// TwinCAT 3 PLC project PLC
// ProgramVersion: 3.1.4024.0
// libraries:
//   SPT Base Types, * (Beckhoff Automation LLC)
//   SPT Components, * (Beckhoff Automation LLC)
//   SPT Motion Control, * (Beckhoff Automation LLC)
//   Tc2_MC2, * (Beckhoff Automation GmbH)
//   Tc2_MC2_Drive, * (Beckhoff Automation GmbH)
//   Tc2_Standard, * (Beckhoff Automation GmbH)
//   Tc2_System, * (Beckhoff Automation GmbH)
//   Tc3_Module, * (Beckhoff Automation GmbH)
//   Tc3_PackML_V2, * (Beckhoff Automation GmbH)
//   VisuDialogs, * (System)
// project tree:
//   / GlobalTextList.TcGTLO, PlcTask.TcTTO, Visualization Manager.TcVMO (not stored)
//   POUs/ MAIN.TcPOU
//   VISUs/ VIS_Main.TcVIS (not stored)
//   _Machine/00_Machine/ FB_UM_Machine.TcPOU
//   _Machine/VISUs/VFMs/ VFM_Machine.TcVIS (not stored), VFM_MachineControl.TcVIS (not stored), VFM_Module.TcVIS (not stored), VFM_OperatingMode.TcVIS (not stored), VFM_PackML.TcVIS (not stored), VFM_PackML_Manual.TcVIS (not stored)
//   _Machine/_Components/Drives/AX5000/ FB_Drive_AX5000.TcPOU, I_Drive_AX5000.TcIO
//   _Machine/_Components/Misc/ FB_StatFilter.TcPOU (not stored), F_TaskTime.TcPOU (not stored)
//   _Machine/_Components/TempController/DUTs/ ST_HMI_TempController.TcDUT (not stored), ST_HMI_TempController_Command.TcDUT (not stored), ST_HMI_TempController_Config.TcDUT (not stored), ST_HMI_TempController_Status.TcDUT (not stored), ST_Param_TempController.TcDUT (not stored)
//   _Machine/_Components/TempController/ FB_TempController.TcPOU, FB_TempCtrl.TcPOU (not stored), I_TemperatureController.TcIO (not stored)
//   _Machine/_Components/TempController/VISUs/VFMs/ VFM_TempController.TcVIS (not stored)
//   _Machine/_Components/TempController/VISUs/ VIS_TempCtrl.TcVIS (not stored)
// real-time tasks:
//   TASK PlcTask: cycle T#10ms, priority 20, ADS port 350
// motion (NC):
//   TASK NC-Task 1 SAF: cycle T#2ms, priority 4, ADS port 501
//   TASK NC-Task 1 SVB: cycle T#10ms, priority 8, ADS port 511
//   AXIS Axis 1 (id 1)
//     OtherSettings: AllowMotionCmdToSlave=true
//     encoder EncType=8
//       EncPara: MaxCount=#x0036ee7f
//     drive DrvType=9
//       DrvPara: MaxCount=#xffffffff, DriveControlDWord=#x00000100
//         Analog: VeloScale=6, TorqueSetpointScale=10, ScaleFactorActTorque=0.1
//         TimeComp: TaskDelayCycles=1
//     controller CtrType=1
//       CtrPara: PriorControlFactor=1
//         Observer: BandWidth=20

CONFIGURATION PLC
    RESOURCE PLC ON TwinCAT3
        TASK PlcTask(INTERVAL := T#10ms, PRIORITY := 20);
        PROGRAM MAIN WITH PlcTask : MAIN;
    END_RESOURCE
END_CONFIGURATION

// ---- _Machine/_Components/Drives/AX5000/I_Drive_AX5000.TcIO
INTERFACE I_Drive_AX5000

METHOD DriveReset : BOOL
VAR_INPUT
END_VAR
END_METHOD

PROPERTY REF_Axis : REFERENCE TO AXIS_REF
GET
END_GET
SET
END_SET
END_PROPERTY

PROPERTY SercosErrorID : UINT
GET
END_GET
END_PROPERTY

END_INTERFACE

// ---- POUs/MAIN.TcPOU
PROGRAM MAIN
VAR
END_VAR

END_PROGRAM

// ---- _Machine/00_Machine/FB_UM_Machine.TcPOU
FUNCTION_BLOCK FB_UM_Machine EXTENDS FB_PackML_BaseModule
VAR
	// Submodules
	
	// Components
	
	// Module Data
	// --Param
	// --Recipe
	// --HMI
	HMI: ST_HMI_Machine;
	
	// Alarms
	
	// Other I/O

	// Machine Control
	rtrigControl: R_TRIG;
	CheckAbort: BOOL;
	CheckStop: BOOL;
	
	// Miscellaneous
	
END_VAR

METHOD PROTECTED Aborted
VAR_INPUT
END_VAR
END_METHOD

METHOD PROTECTED Aborting
VAR_INPUT
END_VAR
CASE _CurrentMode OF
	E_PMLUnitMode.ePMLUnitMode_Production:
        CASE DescendantSequenceState OF
			0:
				NoStateTasksToComplete := FALSE;
				DescendantSequenceState := DescendantSequenceState + 10;
			10:
				StateTasksComplete := TRUE;
		END_CASE
		
	E_PMLUnitMode.ePMLUnitMode_Manual, E_PMLUnitMode.ePMLUnitMode_Maintenance:
        ;	
END_CASE

// Call Super
SUPER^.Aborting();
END_METHOD

METHOD PROTECTED Clearing
VAR_INPUT
END_VAR
CASE _CurrentMode OF
	E_PMLUnitMode.ePMLUnitMode_Production:
        CASE DescendantSequenceState OF
			0:
				NoStateTasksToComplete := FALSE;
				DescendantSequenceState := DescendantSequenceState + 10;
			10:
				StateTasksComplete := TRUE;
		END_CASE
		
	E_PMLUnitMode.ePMLUnitMode_Manual, E_PMLUnitMode.ePMLUnitMode_Maintenance:
        ;	
END_CASE

// Call Super
SUPER^.Clearing();
END_METHOD

METHOD PROTECTED Complete
VAR_INPUT
END_VAR
END_METHOD

//! @summary Initializes event function blocks using this module's name
METHOD PROTECTED CreateEvents

//! @description This method is called by <c>Initialize()</c> as required
// Add your event creation here

// Super call to base
SUPER^.CreateEvents();
END_METHOD

METHOD CyclicLogic
VAR_INPUT
END_VAR
IF NOT _InitComplete THEN
    _InitComplete := Initialize();
    RETURN;
END_IF

MachineControl();

SUPER^.CyclicLogic();
END_METHOD

METHOD PROTECTED Execute
VAR_INPUT
END_VAR
CASE _CurrentMode OF
	E_PMLUnitMode.ePMLUnitMode_Production:
        CASE DescendantSequenceState OF
			0:
				DescendantSequenceState := DescendantSequenceState + 10;
			10:
				;
		END_CASE
		
	E_PMLUnitMode.ePMLUnitMode_Manual, E_PMLUnitMode.ePMLUnitMode_Maintenance:
        ;	
END_CASE
END_METHOD

METHOD PROTECTED Held
VAR_INPUT
END_VAR
END_METHOD

METHOD PROTECTED Holding
VAR_INPUT
END_VAR
CASE _CurrentMode OF
	E_PMLUnitMode.ePMLUnitMode_Production:
        CASE DescendantSequenceState OF
			0:
				NoStateTasksToComplete := FALSE;
				DescendantSequenceState := DescendantSequenceState + 10;
			10:
				StateTasksComplete := TRUE;
		END_CASE
		
	E_PMLUnitMode.ePMLUnitMode_Manual, E_PMLUnitMode.ePMLUnitMode_Maintenance:
        ;	
END_CASE

// Call Super
SUPER^.Holding();
END_METHOD

METHOD PROTECTED Idle
VAR_INPUT
END_VAR
END_METHOD

//! @summary Basic module initialization logic
METHOD PROTECTED Initialize : BOOL;
VAR
	i						 : UDINT;
	varInfo					 : __SYSTEM.VAR_INFO;
	AllSubUnitsInitialized	 : BOOL := TRUE;
	AllComponentsInitialized : BOOL := TRUE;
END_VAR

//! @description This method is called by <c>CyclicLogic()</c> as required
Initialize := FALSE;
CASE DescendantSequenceState OF
    0: // Initialize
        _LogModeChanges         := FALSE;
        _LogStateChanges        := FALSE;
        DescendantSequenceState := DescendantSequenceState + 10;
	
	10: // Register Submodules
		DescendantSequenceState := DescendantSequenceState + 10;
		
    20: // Register Components
		RegisterComponent(TempController);
        DescendantSequenceState := DescendantSequenceState + 10;
		
    30: // Call the Super
        IF SUPER^.Initialize() THEN
            DescendantSequenceState := DescendantSequenceState + 10;
        END_IF
    40:
        Initialize := TRUE;
END_CASE
END_METHOD

METHOD MachineControl
VAR_INPUT
END_VAR
// Control Triggers
rtrigControl(CLK:= HMI.Command.Start XOR HMI.Command.Stop XOR HMI.Command.Reset XOR HMI.Command.Abort);

CASE CurrentState OF
	E_PMLState.ePMLState_Aborting:
		CheckAbort := FALSE;
		CheckStop := FALSE;
		
	E_PMLState.ePMLState_Aborted:
		// Wait for Reset to Clear
		IF rtrigControl.Q AND HMI.Command.Reset THEN
			ChangeState(E_PMLCommand.ePMLCommand_Clear);
		END_IF
		
	E_PMLState.ePMLState_Clearing:
		CheckAbort := TRUE;
		CheckStop := FALSE;
		
	E_PMLState.ePMLState_Stopping:
		CheckAbort := TRUE;
		CheckStop := FALSE;
		
	E_PMLState.ePMLState_Stopped:
		// Wait for Reset
		IF rtrigControl.Q AND HMI.Command.Reset THEN
			ChangeState(E_PMLCommand.ePMLCommand_Reset);
		END_IF
		
	E_PMLState.ePMLState_Resetting:
		CheckAbort := TRUE;
		CheckStop := TRUE;
	
	E_PMLState.ePMLState_Idle:
		// Wait for Start
		IF rtrigControl.Q AND HMI.Command.Start THEN
			ChangeState(E_PMLCommand.ePMLCommand_Start);
		END_IF
	
END_CASE

// Check for Abort or Stop
IF rtrigControl.Q AND HMI.Command.Abort THEN
	ChangeState(E_PMLCommand.ePMLCommand_Abort);
ELSIF rtrigControl.Q AND HMI.Command.Stop THEN
	ChangeState(E_PMLCommand.ePMLCommand_Stop);
END_IF
END_METHOD

METHOD PROTECTED Resetting
VAR_INPUT
END_VAR
CASE _CurrentMode OF
	E_PMLUnitMode.ePMLUnitMode_Production:
        CASE DescendantSequenceState OF
			0:
				NoStateTasksToComplete := FALSE;
				DescendantSequenceState := DescendantSequenceState + 10;
			10:
				StateTasksComplete := TRUE;
		END_CASE
		
	E_PMLUnitMode.ePMLUnitMode_Manual, E_PMLUnitMode.ePMLUnitMode_Maintenance:
        ;	
END_CASE

// Call Super
SUPER^.Resetting();
END_METHOD

METHOD PROTECTED Starting
VAR_INPUT
END_VAR
CASE _CurrentMode OF
	E_PMLUnitMode.ePMLUnitMode_Production:
        CASE DescendantSequenceState OF
			0:
				NoStateTasksToComplete := FALSE;
				DescendantSequenceState := DescendantSequenceState + 10;
			10:
				StateTasksComplete := TRUE;
		END_CASE
		
	E_PMLUnitMode.ePMLUnitMode_Manual, E_PMLUnitMode.ePMLUnitMode_Maintenance:
        ;	
END_CASE

// Call Super
SUPER^.Starting();
END_METHOD

METHOD PROTECTED Stopped
VAR_INPUT
END_VAR
END_METHOD

METHOD PROTECTED Stopping
VAR_INPUT
END_VAR
CASE _CurrentMode OF
	E_PMLUnitMode.ePMLUnitMode_Production:
        CASE DescendantSequenceState OF
			0:
				NoStateTasksToComplete := FALSE;
				DescendantSequenceState := DescendantSequenceState + 10;
			10:
				StateTasksComplete := TRUE;
		END_CASE
		
	E_PMLUnitMode.ePMLUnitMode_Manual, E_PMLUnitMode.ePMLUnitMode_Maintenance:
        ;	
END_CASE

// Call Super
SUPER^.Stopping();
END_METHOD

METHOD PROTECTED Suspended
VAR_INPUT
END_VAR
END_METHOD

METHOD PROTECTED Suspending
VAR_INPUT
END_VAR
CASE _CurrentMode OF
	E_PMLUnitMode.ePMLUnitMode_Production:
        CASE DescendantSequenceState OF
			0:
				NoStateTasksToComplete := FALSE;
				DescendantSequenceState := DescendantSequenceState + 10;
			10:
				StateTasksComplete := TRUE;
		END_CASE
		
	E_PMLUnitMode.ePMLUnitMode_Manual, E_PMLUnitMode.ePMLUnitMode_Maintenance:
        ;	
END_CASE

// Call Super
SUPER^.Suspending();
END_METHOD

METHOD PROTECTED Undefined
VAR_INPUT
END_VAR
END_METHOD

METHOD PROTECTED Unholding
VAR_INPUT
END_VAR
CASE _CurrentMode OF
	E_PMLUnitMode.ePMLUnitMode_Production:
        CASE DescendantSequenceState OF
			0:
				NoStateTasksToComplete := FALSE;
				DescendantSequenceState := DescendantSequenceState + 10;
			10:
				StateTasksComplete := TRUE;
		END_CASE
		
	E_PMLUnitMode.ePMLUnitMode_Manual, E_PMLUnitMode.ePMLUnitMode_Maintenance:
        ;	
END_CASE

// Call Super
SUPER^.Unholding();
END_METHOD

METHOD PROTECTED Unsuspending
VAR_INPUT
END_VAR
CASE _CurrentMode OF
	E_PMLUnitMode.ePMLUnitMode_Production:
        CASE DescendantSequenceState OF
			0:
				NoStateTasksToComplete := FALSE;
				DescendantSequenceState := DescendantSequenceState + 10;
			10:
				StateTasksComplete := TRUE;
		END_CASE
		
	E_PMLUnitMode.ePMLUnitMode_Manual, E_PMLUnitMode.ePMLUnitMode_Maintenance:
        ;	
END_CASE

// Call Super
SUPER^.Unsuspending();
END_METHOD

END_FUNCTION_BLOCK

// ---- _Machine/_Components/Drives/AX5000/FB_Drive_AX5000.TcPOU
(*	Sample Code Disclaimer
	All sample code provided by Beckhoff Automation LLC are for illustrative purposes only
	and are provided “as is” and without any warranties, express or implied.
	Actual implementations in applications will vary significantly.
	Beckhoff Automation LLC shall have no liability for, and does not waive any rights in relation to,
	any code samples that it provides or the use of such code samples for any purpose.
*)
FUNCTION_BLOCK FB_Drive_AX5000 EXTENDS FB_ComponentBase IMPLEMENTS I_Drive_AX5000
VAR
	// Properties
	_SercosErrorID: UINT;
	// References
	refAxis: REFERENCE TO AXIS_REF;
	
	// Method Requests
	DriveResetReq: BOOL;
	
	// General
	fbSoEReset: FB_SoEReset;
	
	
	
	{attribute 'hide'}
	DummyAxis	  : AXIS_REF;
	_ErrorSercoID: INT;
END_VAR

METHOD CyclicLogic : BOOL
VAR_INPUT
END_VAR

VAR
	_ErrorSercoID: UINT;
END_VAR
// Call Super
SUPER^.CyclicLogic();

// Drive Reset Request
IF DriveResetReq THEN
	fbSoEReset.Execute := TRUE;
	DriveResetReq := FALSE;
ELSE
	fbSoEReset.Execute := FALSE;
END_IF

// Call AX5000 SERCOS Reset
fbSoEReset(Axis:= refAxis);

// Busy Logic
IF NOT fbSoEReset.Busy THEN
	_Busy := FALSE;
END_IF

// Error Logic
IF fbSoEReset.Error THEN
	_Busy := FALSE;
	_Error := TRUE;
	_ErrorID := fbSoEReset.AdsErrId;
	_SercosErrorID := fbSoEReset.SercosErrId;
END_IF
END_METHOD

METHOD DriveReset : BOOL
// Call Super
SUPER^.Reset();

IF NOT __ISVALIDREF(refAxis) OR _Busy THEN
    RETURN;
END_IF

_Busy        := TRUE;
_Error       := FALSE;
_ErrorID     := 0;
_SercosErrorID := 0;
DriveResetReq := TRUE;

DriveReset := TRUE;
END_METHOD

//! @summary Basic component initialization logic
METHOD PROTECTED Initialize : BOOL;

//! @description This method is called by <c>CyclicLogic()</c> as required
refAxis REF= DummyAxis;

fbSoEReset.Execute := FALSE;

Initialize := SUPER^.Initialize();
END_METHOD

{warning 'add property implementation'}
PROPERTY REF_Axis : REFERENCE TO AXIS_REF
GET
REF_Axis REF= refAxis;
END_GET
SET
refAxis REF= REF_Axis;
END_SET
END_PROPERTY

{warning 'add property implementation'}
PROPERTY SercosErrorID : UINT
GET
SercosErrorID := _SercosErrorID;
END_GET
END_PROPERTY

END_FUNCTION_BLOCK

// ---- _Machine/_Components/TempController/FB_TempController.TcPOU
(*	Sample Code Disclaimer
	All sample code provided by Beckhoff Automation LLC are for illustrative purposes only
	and are provided “as is” and without any warranties, express or implied.
	Actual implementations in applications will vary significantly.
	Beckhoff Automation LLC shall have no liability for, and does not waive any rights in relation to,
	any code samples that it provides or the use of such code samples for any purpose.
*)
FUNCTION_BLOCK FB_TempController EXTENDS FB_ComponentBase IMPLEMENTS I_TemperatureController
VAR	
	// Properties
	_Enabled: BOOL;
		
	// HMI Interface
	HMI: ST_HMI_TempController;
	
	// Hardware Inputs
	//Feedback AT %I*: INT;
	
	// Hardware Outputs
	CtrlOut AT %Q*: INT; // Scaled for HW Output

	// General
	fbTempCtrl: FB_TempCtrl;
	Setpoint: LREAL;
	Feedback: LREAL; // Scaled for HW Input
	ResetPID: BOOL;
	PID_Output: LREAL;
	EnableReq: BOOL;
	DisableReq: BOOL;
	
	// Simulation

END_VAR

VAR PERSISTENT
	Param: ST_Param_TempController;
END_VAR

METHOD CyclicLogic
VAR_INPUT
END_VAR
// Call Super
SUPER^.CyclicLogic();

IF EnableReq THEN
	_Enabled := TRUE;
	EnableReq := FALSE;
	_Busy := TRUE;
ELSIF DisableReq OR Feedback >= Param.MaxTemp THEN
	_Enabled := FALSE;	
	DisableReq := FALSE;
END_IF

// Input Scaling

// Call PID
fbTempCtrl(
	Enable:= _Enabled, 
	Setpoint:= Param.Setpoint, 
	Feedback:= Feedback, 
	MaxTemperature:= Param.MaxTemp, 
	Kp:= Param.Kp,
	Tn:= Param.Tn,
	Tv:= Param.Tv,
	Td:= Param.Td,
	ControlOutput=>PID_Output , 
);

// Method Calls
CyclicLogic_Simulation();
END_METHOD

METHOD CyclicLogic_Simulation
VAR_INPUT
END_VAR
VAR
	rLossRate: LREAL;
	rGainRate: LREAL;
END_VAR
// Simulate Heating Element
rLossRate := (Feedback - 20.0) * 6.0 / 300.0;
rGainRate := BOOL_TO_LREAL(Enabled) * 0.30 * PID_Output;
Feedback 	:= Feedback + (rGainRate - rLossRate) * fbTempCtrl.CycleTime ;
			
IF Feedback < 20.0 THEN
	Feedback := 20.0;
END_IF
END_METHOD

METHOD Disable
VAR_INPUT
END_VAR

VAR
	
END_VAR
// Disable Request
DisableReq := TRUE;
END_METHOD

METHOD Enable
VAR_INPUT
END_VAR

VAR
	
END_VAR
// Enable Request
EnableReq := TRUE;
END_METHOD

PROPERTY Enabled : BOOL
GET
Enabled := _Enabled;
END_GET
END_PROPERTY

//! @summary Provides interlocks for HMI control and updates HMI status information for this component
METHOD PROTECTED HMICommunication

//! @description This method is called cyclically by <c>CyclicLogic()</c>
// Call Super
SUPER^.HMICommunication();

Param := HMI.Config.Param;

// Manual Controls
IF HMI.Command.Manual THEN
	IF _Enabled THEN
		IF HMI.Command.Stop THEN
			Disable();
		END_IF
	ELSE
		IF HMI.Command.Start THEN
			Enable();
		END_IF
	END_IF	
END_IF

// Status Update
HMI.Status.Enabled := _Enabled;
HMI.Status.CtrlOutput := PID_Output;
HMI.Status.Actual := Feedback;
END_METHOD

//! @summary Basic component initialization logic
METHOD PROTECTED Initialize : BOOL;

//! @description This method is called by <c>CyclicLogic()</c> as required
IF fbTempCtrl.CycleTime = 0.0 THEN
	fbTempCtrl.CycleTime := F_TaskTime();
END_IF

HMI.Config.Param := Param;

//Call base class Initialize
Initialize := SUPER^.Initialize();
END_METHOD

METHOD Manual
VAR_INPUT
	ManualMode: bool;
END_VAR
HMI.Command.Manual := ManualMode;
END_METHOD

END_FUNCTION_BLOCK

// ---- GlobalTextList.TcGTLO
TEXTLIST GlobalTextList
  672 = '%3.1f %%'
  685 = '%s'
  680 = 'Abort'
  11 = 'Aborted'
  86 = 'Aborting'
  452 = 'Clear'
  467 = 'Clearing'
  754 = 'Complete'
  302 = 'Completing'
  663 = 'Execute'
  51 = 'Held'
  744 = 'Hold'
  369 = 'Holding'
  236 = 'I'
  342 = 'Idle'
  46 = 'Maintenance'
  904 = 'Manual'
  820 = 'O'
  929 = 'Production'
  263 = 'PV: %3.1f'
  799 = 'R'
  181 = 'Reset'
  123 = 'Resetting'
  639 = 'SC'
  77 = 'Start'
  888 = 'Starting'
  516 = 'State: %s'
  828 = 'Stop'
  796 = 'Stopped'
  161 = 'Stopping'
  806 = 'Suspend'
  623 = 'Suspended'
  229 = 'Suspending'
  304 = 'SV: %3.1f'
  124 = 'Temp Controller'
  782 = 'Un-Hold'
  466 = 'Un-Holding'
  901 = 'Un-Suspend'
  254 = 'Un-Suspending'
  197 = 'Unhold'
  832 = 'Unsuspend'
END_TEXTLIST
